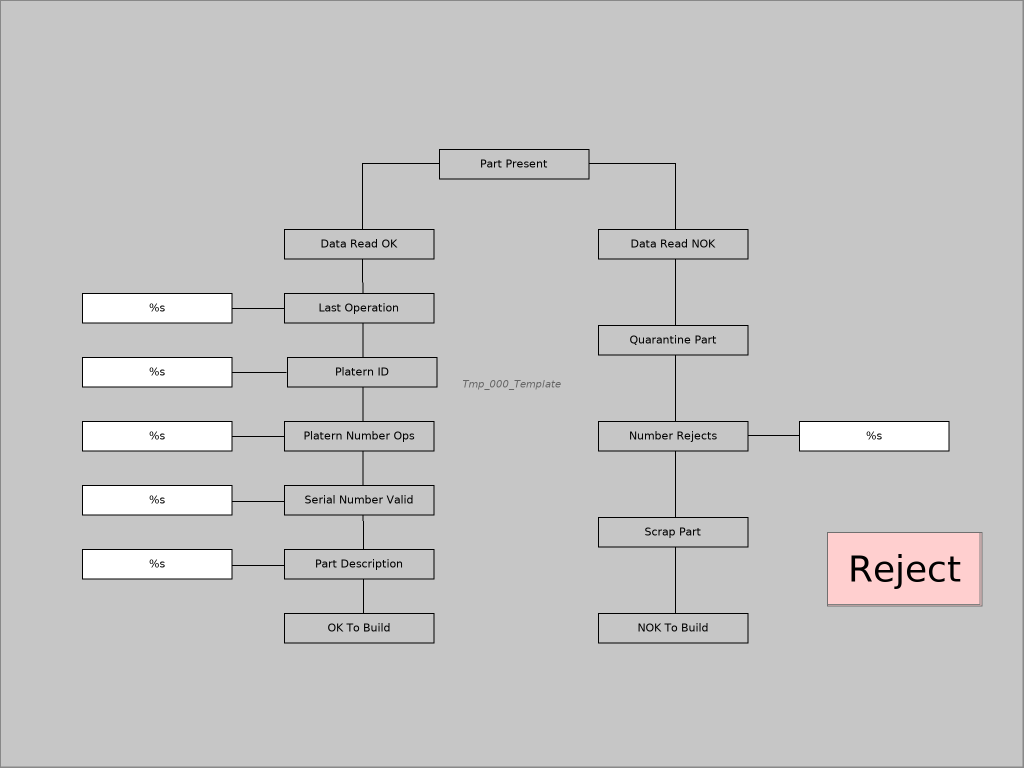
VISUALIZATION Prc_500_Part  // 1024x768
    Frame (0,0 1024x768)
        shows Tmp_000_Template(header := gHMIData.hmiHeader)
    Line (362,163) (675,163)
    Line (747,435) (803,435)
    Line (230,308) (286,308)
    Line (230,372) (286,372)
    Line (230,436) (286,436)
    Line (229,501) (285,501)
    Line (229,565) (285,565)
    Line (675,163) (675,640)
    Line (362,163) (363,640)
    Rectangle (284,421 150x30), "Platern Number Ops", colour toggle: Mc_Global.part.PlaternNumOpsValid
    Rectangle (287,357 150x30), "Platern ID", colour toggle: Mc_Global.part.PlaternIDValid
    Rectangle (284,229 150x30), "Data Read OK", colour toggle: Mc_Global.part.DataReadOK
    Rectangle (598,229 150x30), "Data Read NOK", colour toggle: Mc_Global.part.DataReadNOK
    Rectangle (284,485 150x30), "Serial Number Valid", colour toggle: Mc_Global.part.SerialNumberValid
    Rectangle (284,549 150x30), "Part Description", colour toggle: Mc_Global.part.PartDescriptionValid
    Rectangle (284,613 150x30), "OK To Build", colour toggle: Mc_Global.part.OKtoBuild
    Rectangle (598,613 150x30), "NOK To Build", colour toggle: Mc_Global.part.NOKtoBuild
    Rectangle (598,325 150x30), "Quarantine Part", colour toggle: Mc_Global.part.QuarantinePart
    Rectangle (598,517 150x30), "Scrap Part", colour toggle: Mc_Global.part.ScrapPart
    Rectangle (598,421 150x30), "Number Rejects", colour toggle: Mc_Global.part.NumberOfRejectAttemptsFailed
    Rectangle (284,293 150x30), "Last Operation", colour toggle: Mc_Global.part.LastOperationNumberValid
    Rectangle (82,485 150x30), "%s", text variable: Mc_Global.part.SerialNumber
    Rectangle (82,421 150x30), "%s", text variable: Mc_Global.part.PlaternNumOps
    Rectangle (82,357 150x30), "%s", text variable: Mc_Global.part.PlaternID
    Rectangle (82,293 150x30), "%s", text variable: Mc_Global.part.LastOperationNumber
    Rectangle (82,549 150x30), "%s", text variable: Mc_Global.part.PartDescription
    Rectangle (799,421 150x30), "%s", text variable: Mc_Global.part.NumberOfRejectAttempts
    Rectangle (439,149 150x30), "Part Present", colour toggle: Mc_Global.part.PartPresent
    Button (827,532 155x74), "Reject"
        OnMouseClick: OpenDialog Dialog=dialogReject, OpenModal=True, OpenCentered=True
END_VISUALIZATION

(* stored: Version 1.1.0.1, ProductVersion 3.1.4024.12
   Visu Prc_500_Part: Id {01a3fd68-7c4e-41ec-a83c-7689ac5914e7} *)
